INTERFACE I_Motor1R

PROPERTY P_Laufzeit : TIME
GET
END_GET
END_PROPERTY

PROPERTY P_MaxDrz : INT
SET
END_SET
END_PROPERTY

END_INTERFACE

(* stored: Version 1.1.0.1, ProductVersion 3.1.4024.12
   Itf I_Motor1R: Id {b2f9a347-f0d3-4207-b300-f309dfcbc50c}
   Property P_Laufzeit: Id {07a4ec4a-20e2-448f-9eb9-349f5871142f}
   Get Get: Id {7c640eb3-ade5-47ec-a7d0-ba29cc386d5c}
   Property P_MaxDrz: Id {e89f8272-13df-449e-85fc-984eb699f2cd}
   Set Set: Id {0dffa0f3-67f5-4858-9446-ac5a79509cf5} *)
